Staubli VAL3: .pjx

--- .pjx ---
Parameters version=s7.11.3 stackSize=5000 millimeterUnit=true
Program file=getNum.pgx
Program file=init.pgx
Program file=start.pgx
Program file=stop.pgx
Program file=tPosition.pgx
Program file=tCommande.pgx
Program file=tRobot.pgx
Data file=numericalTwins.dtx

--- .dtx ---
mdesc mNomSpeed
sio sioSocket = {link=Socket\toto}
string sTaskPos
string sTaskCmd
string sTaskRobot
jointRx jHere
string sData
num nFrameIndex
num nEol
bool bOvrPosition
num nOvrPos
num nPrevOvrPos
num nSof
num nEof
num nDivider
num nNbChar
num nData
string sDataIn
bool bResult
pointRx pCmdQueue[5]
  [0] = {fatherId=world[0]}
  [1] = {fatherId=world[0]}
  [2] = {fatherId=world[0]}
  [3] = {fatherId=world[0]}
  [4] = {fatherId=world[0]}
num nTypeQueue[5]
num nIndexQueue[5]
num nVelQueue[5]
num nQueueWrite
num nQueueRead
num nQueueCount
num nQueueSize
num nCmdIndex
num nCmdType
num nCmdVel
num nLastIndex
bool bFinish
jointRx jStart
string sAck
num nAckIndex

--- numericalTwins.dtx ---
bool bFinish
bool bOvrPosition
bool bResult = true
frame fPlateau = {x=632.308207, y=706.981098, z=-559.699722, rx=-0.00630742, ry=-0.102848, rz=-0.154308, fatherId=world[0]}
jointRx home = {j1=64, j2=-30, j3=143, j4=-103, j5=60, j6=116}
jointRx jHere = {j1=45.383273, j2=1.666947, j3=107.278201, j4=-97.512292, j5=76.926774, j6=121.888458}
jointRx jStart
mdesc mNomSpeed = {vel=50}
mdesc vitextrusion = {rmax=500, tmax=17, leave=15, reach=15}
num nAckIndex
num nCmdIndex = 4
num nCmdType = 1
num nCmdVel = 50
num nData = 10
num nDivider = 59
num nEof = 125
num nEol = 10
num nFrameIndex = 3553
num nIndexQueue[5]
  [0] = 1
  [1] = 2
  [2] = 3
  [3] = 4
num nLastIndex
num nNbChar
num nOvrPos
num nPrevOvrPos
num nQueueCount
num nQueueRead
num nQueueSize = 5
num nQueueWrite
num nSof = 123
num nTypeQueue[5]
  [0] = 1
  [1] = 1
  [2] = 1
  [3] = 1
num nVelQueue[5]
  [0] = 50
  [1] = 50
  [2] = 50
  [3] = 50
pointRx pAccostage = {x=200, y=-150, z=5, rx=-180, ry=7.016478e-15, rz=-180, fatherId=fPlateau[0]}
pointRx pChauffe = {x=-200, z=200, ry=180, fatherId=fPlateau[0]}
pointRx pCmdQueue[5]
  [0] = {x=371.256502, y=762.70159, z=186.0845966, rx=89.692992, ry=69.84956, rz=-90.0731633, shoulder=lefty, elbow=epositive, wrist=wpositive, fatherId=world[0]}
  [1] = {x=371.256502, y=762.70159, z=186.0845966, rx=89.692992, ry=69.84956, rz=-90.0731633, shoulder=lefty, elbow=epositive, wrist=wpositive, fatherId=world[0]}
  [2] = {x=371.256502, y=762.70159, z=186.0845966, rx=89.692992, ry=69.84956, rz=-90.0731633, shoulder=lefty, elbow=epositive, wrist=wpositive, fatherId=world[0]}
  [3] = {x=371.256502, y=762.70159, z=186.0845966, rx=89.692992, ry=69.84956, rz=-90.0731633, shoulder=lefty, elbow=epositive, wrist=wpositive, fatherId=world[0]}
  [4] = {x=371.256502, y=762.70159, z=186.0845966, rx=89.692992, ry=69.84956, rz=-90.0731633, shoulder=lefty, elbow=epositive, wrist=wpositive, fatherId=world[0]}
pointRx pDegagement = {z=200, ry=180, fatherId=fPlateau[0]}
pointRx pHere = {x=832.0401931, y=692.000932864, z=529.509333, rx=84.591408, ry=60.0803316, rz=-73.577687, shoulder=lefty, elbow=epositive, wrist=wpositive, fatherId=world[0]}
sio sioSocket = {link=Socket\toto}
string sAck
string sData = "{3553;    45.383;     1.667;   107.278;   -97.512;    76.927;   121.888;832.04 ;692.001;529.509;84.591;60.08 ;-73.578}"
string sDataIn
string sTaskCmd = "tCommande"
string sTaskPos = "tPosition"
string sTaskRobot = "tRobot"
tool tBuse = {x=551, y=-30, z=75, ry=90, rz=-20, fatherId=flange[0], ioLink=valve1}
tool tPalpage = {x=655.7, y=-30, z=75, ry=90, rz=-20, fatherId=flange[0]}

--- start.pgx ---
program start()
begin
  // Initialisation
  call init()

  // tPosition : envoi position toutes les 40ms (sync)
  taskCreateSync sTaskPos,0.04,bOvrPosition,tPosition()
  wait(taskStatus(sTaskPos)==1)

  // Mouvement vers le point de test avec l'outil Buse
  movej(home,tBuse,vitextrusion)
  waitEndMove()

  // D├⌐finition du point de d├⌐gagement et d'accostage
  // Vous pouvez d├⌐finir pDegagement en dur ici ou l'avoir appris manuellement
  // pAccostage.trsf.z = nHcouche1
  //pAccostage.trsf={200,-150,nHcouche1,0,180,0}
  // --- Ex├⌐cution ---
  // Demarrage de l extrusion
  movel(pChauffe,tBuse,vitextrusion)
  waitEndMove()
  // 1. Approche
  movel(pAccostage,tBuse,vitextrusion)
  waitEndMove()



  // tCommande : reception des commandes
  taskCreate sTaskCmd,100,tCommande()
  wait(taskStatus(sTaskCmd)==1)

  // tRobot : execution des mouvements
  taskCreate sTaskRobot,100,tRobot()
  wait(taskStatus(sTaskRobot)==1)

  // Surveillance des overruns
  while true
    if nPrevOvrPos!=nOvrPos
      logMsg("Overrun dans la tache "+sTaskPos)
      nPrevOvrPos=nOvrPos
    endIf
    delay(0)
  endWhile


  waitEndMove()

  // 3. Repli
  movel(pDegagement,tBuse,vitextrusion)
  movel(pChauffe,tBuse,vitextrusion)

  waitEndMove()


end

--- getNum.pgx ---
program getNum(num& x_nNum (dimensions=1), num x_nEnd (dimensions=1))
begin
  sDataIn=""
  do
    nNbChar=sioGet(sioSocket,nData)
    if nNbChar>0 and nData!=x_nEnd
      sDataIn=sDataIn+chr(nData)
    endIf
  until nNbChar>0 and nData==x_nEnd
  sDataIn=toNum(sDataIn,x_nNum,bResult)
end

--- init.pgx ---
program init()
begin
  // Noms des taches
  sTaskPos="tPosition"
  sTaskCmd="tCommande"
  sTaskRobot="tRobot"

  // Overrun
  bOvrPosition=false
  nOvrPos=0
  nPrevOvrPos=0

  // Index trames emises
  nFrameIndex=0

  // Caracteres de protocole
  nEol=10
  nSof=asc("{",0)
  nEof=asc("}",0)
  nDivider=asc(";",0)

  // File circulaire
  nQueueSize=5
  nQueueWrite=0
  nQueueRead=0
  nQueueCount=0

  // Flags
  bFinish=false
  nLastIndex=0

  // Initialisation file avec repere world
  pCmdQueue[0]=here(flange,world)
  pCmdQueue[1]=here(flange,world)
  pCmdQueue[2]=here(flange,world)
  pCmdQueue[3]=here(flange,world)
  pCmdQueue[4]=here(flange,world)

  // Socket TCP
  sioCtrl(sioSocket,"port",2005)
  sioCtrl(sioSocket,"target","192.168.99.6")
  sioCtrl(sioSocket,"endOfString",nEol)
  sioCtrl(sioSocket,"timeout",-1)
  sioCtrl(sioSocket,"nagle",false)
end

--- tCommande.pgx ---
program tCommande()
begin
  // Trame attendue depuis le PC :
  // {index;type;x;y;z;rx;ry;rz;vel}
  // type : 0=movej, 1=movel
  // vel  : vitesse TCP mm/s

  while true
    // Attente que la file ne soit pas pleine
    wait(nQueueCount<nQueueSize)

    // Recherche debut de trame
    do
      nNbChar=sioGet(sioSocket,nData)
    until nNbChar>0 and nData==nSof

    // Lecture des 9 champs
    call getNum(nCmdIndex,nDivider)
    call getNum(nCmdType,nDivider)
    call getNum(pCmdQueue[nQueueWrite].trsf.x,nDivider)
    call getNum(pCmdQueue[nQueueWrite].trsf.y,nDivider)
    call getNum(pCmdQueue[nQueueWrite].trsf.z,nDivider)
    call getNum(pCmdQueue[nQueueWrite].trsf.rx,nDivider)
    call getNum(pCmdQueue[nQueueWrite].trsf.ry,nDivider)
    call getNum(pCmdQueue[nQueueWrite].trsf.rz,nDivider)
    call getNum(nCmdVel,nEof)

    // Ecriture dans la file
    nTypeQueue[nQueueWrite]=nCmdType
    nIndexQueue[nQueueWrite]=nCmdIndex
    nVelQueue[nQueueWrite]=nCmdVel

    // Avance le pointeur d ecriture (circulaire)
    nQueueWrite=nQueueWrite+1
    if nQueueWrite>=nQueueSize
      nQueueWrite=0
    endIf
    nQueueCount=nQueueCount+1

    delay(0)
  endWhile
end

--- tPosition.pgx ---
program tPosition()
  local num l_nIndex
begin
  // Trame envoy├⌐e au PC :
  // {index;j1;j2;j3;j4;j5;j6;x;y;z;rx;ry;rz}
  // Une seule paire d'accolades, 13 champs s├⌐par├⌐s par ";"

  while true
    delay(0)

    nFrameIndex=nFrameIndex+1

    // Position articulaire courante
    jHere=herej()
    // Position cartesienne courante
    pHere=here(flange,world)

    // Construction de la trame (128 caract├¿res max)
    sData="{"
    sData=sData+toString("",nFrameIndex)+";"
    sData=sData+toString("10.3",jHere.j1)+";"
    sData=sData+toString("10.3",jHere.j2)+";"
    sData=sData+toString("10.3",jHere.j3)+";"
    sData=sData+toString("10.3",jHere.j4)+";"
    sData=sData+toString("10.3",jHere.j5)+";"
    sData=sData+toString("10.3",jHere.j6)+";"
    sData=sData+toString(".3",pHere.trsf.x)+";"
    sData=sData+toString(".3",pHere.trsf.y)+";"
    sData=sData+toString(".3",pHere.trsf.z)+";"
    sData=sData+toString(".3",pHere.trsf.rx)+";"
    sData=sData+toString(".3",pHere.trsf.ry)+";"
    sData=sData+toString(".3",pHere.trsf.rz)+"}"

    // Envoi octet par octet
    for l_nIndex=0 to len(sData)-1
      sioSet(sioSocket,asc(sData,l_nIndex))
    endFor
    // Fin de trame LF
    sioSet(sioSocket,nEol)

    // D├⌐tection overrun
    if bOvrPosition
      nOvrPos=nOvrPos+1
    endIf
  endWhile
end

--- tRobot.pgx ---
program tRobot()
  local num l_nIdx
begin

  while !bFinish
    // Attente qu il y ait au moins un point dans la file
    wait(nQueueCount > 0)

    // Lecture du point courant dans la file
    l_nIdx = nQueueRead

    // Verification continuite des trames
    if nIndexQueue[l_nIdx] == nLastIndex + 1

      // Configuration vitesse pour ce point
      mNomSpeed.vel = nVelQueue[l_nIdx]
      pCmdQueue[l_nIdx].config.shoulder = lefty
      pCmdQueue[l_nIdx].config.wrist    = wpositive
      pCmdQueue[l_nIdx].config.elbow    = epositive
      logMsg("Point: x=" + toString(".1", pCmdQueue[l_nIdx].trsf.x) + " y=" + toString(".1", pCmdQueue[l_nIdx].trsf.y) + " z=" + toString(".1", pCmdQueue[l_nIdx].trsf.z))

      // Execution du mouvement selon le type
      if nTypeQueue[l_nIdx] == 0
        movel(pCmdQueue[l_nIdx], tBuse, mNomSpeed)
      else
        movel(pCmdQueue[l_nIdx], tBuse, mNomSpeed)
      endIf
      waitEndMove()

      nLastIndex = nIndexQueue[l_nIdx]

      // Envoi ACK + etat file : {ACK;index_execute;n_restant}
      sAck = "{ACK;" + toString("", nLastIndex) + ";" + toString("", nQueueCount) + "}"
      nAckIndex = 0
      while nAckIndex < len(sAck)
        sioSet(sioSocket, asc(sAck, nAckIndex))
        nAckIndex = nAckIndex + 1
      endWhile
      sioSet(sioSocket, nEol)

    else
      logMsg("Erreur trame, attendue: " + toString("", nLastIndex+1) + " recue: " + toString("", nIndexQueue[l_nIdx]))
      nLastIndex = nIndexQueue[l_nIdx] - 1
    endIf

    // Avance le pointeur de lecture
    nQueueRead = nQueueRead + 1
    if nQueueRead >= nQueueSize
      nQueueRead = 0
    endIf
    nQueueCount = nQueueCount - 1

    delay(0)
  endWhile

  waitEndMove()
end
